TYPE CmpHMI :
STRUCT
	
	Title : STRING := '';
	Message : STRING := '';
	Timeout : TIME := T#0s;
	InformationOnly :BOOL;
	Trigger : BOOL;
	RespPositive : BOOL;
	RespNegative : BOOL;
	RespTimeout : BOOL;
	HeartbeatOK : BOOL;
	
END_STRUCT
END_TYPE

(* stored: Version 1.1.0.1, ProductVersion 3.1.4024.6
   DUT CmpHMI: Id {616673b7-b8a9-4680-b7f2-91a7a1eba805} *)
